//---------------------------------------------------------------------------------------------------------------
//
//  HAUD 2025.02.24
//
//  - test program
//    - handshakes with process instances
//
//---------------------------------------------------------------------------------------------------------------
PROGRAM PROCESS_HANDSHAKE
VAR_INPUT
  bEnable     : Bool;
END_VAR
VAR
  bInit       : BOOL;

  // singke switches for testing
  bDisableBufferInfeedSender      : BOOL; // this buffer has to be the first to stop feeding movers, since movers must not be waiting in the vertical 180° curve
  bDisableBufferInfeed            : BOOL;
END_VAR

IF NOT binit
THEN
  bInit                                                 := TRUE;

  GVL_APPLICATION.tProcess[E_INSTANCE.INFEED]           := T#600MS;
  GVL_APPLICATION.tProcess[E_INSTANCE.OUTFEED_ROBOT_R1] := T#800MS;
  GVL_APPLICATION.tProcess[E_INSTANCE.OUTFEED_ROBOT_R2] := T#800MS;
END_IF
//-----------------------------------------------------------------------------------
// - SenderBufferInfeed  : 1 XtsStation 
//                    movers are handled when entering position area 
//                    movers are sent to BufferInfeed, so that BufferInfeed has 12 mover ready
//                    movers do stop here, wait until there is room for movers
//                    

CASE GVL_APPLICATION.SenderBufferInfeed.State
OF
  E_INSTANCE_STATE.DISABLED:
    CASE GVL_APPLICATION.SenderBufferInfeed.Progress
    OF
      E_PROGRESS.PROGRESS_BUSY:
        IF bEnable
        THEN
          GVL_APPLICATION.SenderBufferInfeed.Command    := SEL(bDisableBufferInfeedSender, E_INSTANCE_CMD.ENABLE, E_INSTANCE_CMD.DISABLE);
        END_IF
    END_CASE

  E_INSTANCE_STATE.FINISH:
    CASE GVL_APPLICATION.SenderBufferInfeed.Progress
    OF
      E_PROGRESS.PROGRESS_BUSY:
        IF bEnable
        THEN
          GVL_APPLICATION.SenderBufferInfeed.Command    := SEL(bDisableBufferInfeedSender, E_INSTANCE_CMD.FINISH, E_INSTANCE_CMD.DISABLE);
        END_IF
    END_CASE
END_CASE

//-----------------------------------------------------------------------------------
// - BufferInfeed     : single XtsStation which looks for input trigger from transfersystem, 
//                      transfersystem writes positions of XtsStations to be used at Infeed. 
//                      BufferInfeed is writing ItfProcessCollector[BufferInfeed.ProcessTarget].ActivateStation for BufferInfeed target (Infeed / 12 XtsStations).
//                      BufferInfeed sends required amount of movers to WaitPos of XtsStations of BufferInfeed target (Infeed / 12 XtsStations).

CASE GVL_APPLICATION.BufferInfeed.State
OF
  E_INSTANCE_STATE.DISABLED:
    CASE GVL_APPLICATION.BufferInfeed.Progress
    OF
      E_PROGRESS.PROGRESS_BUSY:
        IF bEnable
        THEN
          GVL_APPLICATION.BufferInfeed.Command          := E_INSTANCE_CMD.ENABLE;
        END_IF
    END_CASE

  E_INSTANCE_STATE.FINISH:
    CASE GVL_APPLICATION.BufferInfeed.Progress
    OF
      E_PROGRESS.PROGRESS_OCCUPIED:
        IF bEnable
        THEN
          GVL_APPLICATION.BufferInfeed.Command          := E_INSTANCE_CMD.PROCEED;
        END_IF
    END_CASE
END_CASE


//-----------------------------------------------------------------------------------
// - Infeed         : 12 XtsStations for transfersystem to unload
//                    Infeed is pulling in the movers according to list entry from BufferInfeed
//                    one stop only
//                    must be checked for all mover standstill in PosStop[1] of each XtsStation
//                    must be released by handshake from transfersystem (this is done by a TON for now)

CASE GVL_APPLICATION.Infeed.State
OF
  E_INSTANCE_STATE.DISABLED:
    CASE GVL_APPLICATION.Infeed.Progress
    OF
      E_PROGRESS.PROGRESS_BUSY:
        IF bEnable
        THEN
          GVL_APPLICATION.Infeed.Command                := E_INSTANCE_CMD.ENABLE;
        END_IF
    END_CASE

  E_INSTANCE_STATE.WORKING:
    CASE GVL_APPLICATION.Infeed.Progress
    OF
      E_PROGRESS.PROGRESS_BUSY:
        GVL_APPLICATION.tonProcess [E_INSTANCE.INFEED]
                                            (IN         := FALSE, 
                                             PT         := GVL_APPLICATION.tProcess[E_INSTANCE.INFEED]);
        IF bEnable
        THEN
          GVL_APPLICATION.Infeed.Command                := E_INSTANCE_CMD.WORK;
        END_IF


      E_PROGRESS.PROGRESS_CHECK:
        GVL_APPLICATION.tonProcess [E_INSTANCE.INFEED]
                                            (IN         := TRUE, 
                                             PT         := GVL_APPLICATION.tProcess[E_INSTANCE.INFEED]);

        IF GVL_APPLICATION.tonProcess [E_INSTANCE.INFEED].Q
        THEN
          IF bEnable
          THEN
            GVL_APPLICATION.Infeed.Command              := E_INSTANCE_CMD.FINISH;
          END_IF
        END_IF
    END_CASE
END_CASE


//-----------------------------------------------------------------------------------
// - BufferOutfeedRobot  : single XtsStation which distributes movers to OutfeedR2 and OutfeedR1 
//                    Infeed sends all movers here 
//                    BufferOutfeed ensures that OutputR2 and OutputR1 have 12 movers each for every job
//                    BufferOutfeed checks if the Queue of this single XtsStation is empty or not

CASE GVL_APPLICATION.BufferOutfeedRobot.State
OF
  E_INSTANCE_STATE.DISABLED:
    CASE GVL_APPLICATION.BufferOutfeedRobot.Progress
    OF
      E_PROGRESS.PROGRESS_BUSY:
        IF bEnable
        THEN
          GVL_APPLICATION.BufferOutfeedRobot.Command    := E_INSTANCE_CMD.ENABLE;
        END_IF
    END_CASE

  E_INSTANCE_STATE.FINISH:
    CASE GVL_APPLICATION.BufferOutfeedRobot.Progress
    OF
      E_PROGRESS.PROGRESS_BUSY:
        IF bEnable
        THEN
          GVL_APPLICATION.BufferOutfeedRobot.Command    := E_INSTANCE_CMD.FINISH;
        END_IF
    END_CASE
END_CASE


//-----------------------------------------------------------------------------------
// - Outfeed_R1  : 12 XtsStations for Robot 
//                    All XtsStations must be filled before robot can start 
//                    affter process all movers are sent to Sender process (high speed for the way back)
//                     
//                    
(*
CASE GVL_APPLICATION.Outfeed_R1.State
OF
  E_INSTANCE_STATE.DISABLED:
    CASE GVL_APPLICATION.Outfeed_R1.Progress
    OF
      E_PROGRESS.PROGRESS_BUSY:
        GVL_APPLICATION.Outfeed_R1.Command              := E_INSTANCE_CMD.ENABLE;
    END_CASE

  E_INSTANCE_STATE.WORKING:
    CASE GVL_APPLICATION.Outfeed_R1.Progress
    OF
      E_PROGRESS.PROGRESS_BUSY:
        GVL_APPLICATION.tonProcess [E_INSTANCE.OUTFEED_ROBOT_R1]
                                            (IN         := FALSE, 
                                             PT         := GVL_APPLICATION.tProcess[E_INSTANCE.OUTFEED_ROBOT_R1]);
        GVL_APPLICATION.Outfeed_R1.Command              := E_INSTANCE_CMD.WORK;

      E_PROGRESS.PROGRESS_CHECK:
        GVL_APPLICATION.tonProcess [E_INSTANCE.OUTFEED_ROBOT_R1]
                                            (IN         := TRUE, 
                                             PT         := GVL_APPLICATION.tProcess[E_INSTANCE.OUTFEED_ROBOT_R1]);

        IF GVL_APPLICATION.tonProcess [E_INSTANCE.OUTFEED_ROBOT_R1].Q
        THEN
          GVL_APPLICATION.Outfeed_R1.Command            := E_INSTANCE_CMD.FINISH;
        END_IF
    END_CASE
END_CASE
*)

//-----------------------------------------------------------------------------------
// - Outfeed_R2  : 12 XtsStations for Robot 
//                    All XtsStations must be filled before robot can start 
//                    affter process all movers are sent to Sender process (high speed for the way back)
//                     
//                    

CASE GVL_APPLICATION.Outfeed_R2.State
OF
  E_INSTANCE_STATE.DISABLED:
    CASE GVL_APPLICATION.Outfeed_R2.Progress
    OF
      E_PROGRESS.PROGRESS_BUSY:
        IF bEnable
        THEN
          GVL_APPLICATION.Outfeed_R2.Command            := E_INSTANCE_CMD.ENABLE;
          GVL_APPLICATION.Outfeed_R1.Command            := E_INSTANCE_CMD.ENABLE;
        END_IF
    END_CASE

  E_INSTANCE_STATE.WORKING:
    CASE GVL_APPLICATION.Outfeed_R2.Progress
    OF
      E_PROGRESS.PROGRESS_BUSY:
        GVL_APPLICATION.tonProcess [E_INSTANCE.OUTFEED_ROBOT_R2]
                                            (IN         := FALSE, 
                                             PT         := GVL_APPLICATION.tProcess[E_INSTANCE.OUTFEED_ROBOT_R2]);
        IF (GVL_APPLICATION.Outfeed_R1.State = GVL_APPLICATION.Outfeed_R2.State)
        THEN 
          IF bEnable
          THEN
            GVL_APPLICATION.Outfeed_R2.Command          := E_INSTANCE_CMD.WORK;
            GVL_APPLICATION.Outfeed_R1.Command          := E_INSTANCE_CMD.WORK;
          END_IF
        END_IF

      E_PROGRESS.PROGRESS_CHECK:
        GVL_APPLICATION.tonProcess [E_INSTANCE.OUTFEED_ROBOT_R2]
                                            (IN         := TRUE, 
                                             PT         := GVL_APPLICATION.tProcess[E_INSTANCE.OUTFEED_ROBOT_R2]);

        IF GVL_APPLICATION.tonProcess [E_INSTANCE.OUTFEED_ROBOT_R2].Q
        THEN
          IF bEnable
          THEN
            GVL_APPLICATION.Outfeed_R2.Command          := E_INSTANCE_CMD.FINISH;
            GVL_APPLICATION.Outfeed_R1.Command          := E_INSTANCE_CMD.FINISH;
          END_IF
        END_IF
    END_CASE
END_CASE



//-----------------------------------------------------------------------------------
// - SenderFast  : 1 XtsStation 
//                    movers are handled when entering position area 
//                    movers are accelerated to max speed
//                    movers do not stop here
//                    

CASE GVL_APPLICATION.SenderFast.State
OF
  E_INSTANCE_STATE.DISABLED:
    CASE GVL_APPLICATION.SenderFast.Progress
    OF
      E_PROGRESS.PROGRESS_BUSY:
        IF bEnable
        THEN
          GVL_APPLICATION.SenderFast.Command            := E_INSTANCE_CMD.ENABLE;
        END_IF
    END_CASE

  E_INSTANCE_STATE.FINISH:
    CASE GVL_APPLICATION.SenderFast.Progress
    OF
      E_PROGRESS.PROGRESS_BUSY:
        IF bEnable
        THEN
          GVL_APPLICATION.SenderFast.Command            := E_INSTANCE_CMD.FINISH;
        END_IF
    END_CASE
END_CASE

END_PROGRAM

(* stored: Version 1.1.0.1, ProductVersion 3.1.4024.15
   POU PROCESS_HANDSHAKE: Id {db5864b5-04e2-4cc0-83c9-c75fef762d3c}, SpecialFunc None *)
